{attribute 'qualified_only'}
TYPE GetDeviceDataSteps :
(
	Begin,
  FetchDeviceTypes,
  ResetId1,
  GetDeviceNames,
  ResetId2,
  GetDeviceNetIds,
  End
);
END_TYPE

(* stored: Version 1.1.0.1
   DUT GetDeviceDataSteps: Id {7e389f72-6520-46e6-89b4-6fcc0f3eacb7} *)
